Staubli VAL3: setTool.pgx

public program setTool(num x_nIndexGun)
begin
  //
end
